{attribute addProperty BoxType "AX8118-0000-0041-0041"}
{attribute addProperty Id "DeviceDevice_FD48B4B01620Ch_ACh_A_99F8614F240300WcStateAT %I*WcState_98A4DF7520.250InfoDataAT %I*InfoData_F030DC9B200250"}
{attribute addProperty CRC "1708484915"}
{attribute addProperty SizeInBites "458"}
{attribute addProperty SizeInBytes "57.25"}
TYPE AX8118_E3898C73 :
STRUCT
	{attribute addProperty Name "Device"}
	Device : Device_FD48B4B0;
	{attribute addProperty Name "Ch_A"}
	Ch_A : Ch_A_99F8614F;
	{attribute addProperty Name "WcState"}
	WcState : WcState_98A4DF75;
	{attribute addProperty Name "InfoData"}
	InfoData : InfoData_F030DC9B;
END_STRUCT
END_TYPE

(* stored: Version 1.2.0.0, ProductVersion 3.1.4024.9
   DUT AX8118_E3898C73: Id {869cfa1f-35c3-4e88-b4d9-1942c91ae292} *)
